TYPE ST_CoEIndSub :
STRUCT
	nIndex	:	WORD;
	nSubIndex	:	BYTE;
END_STRUCT
END_TYPE

(* stored: Version 1.1.0.1, ProductVersion 3.1.4020.12
   DUT ST_CoEIndSub: Id {d0078caa-6211-47c1-a2ac-3599e1fb4706} *)
